Fanuc KAREL source: kb00086.KL

-- PROVISIONAL review KL for V770-1; original PC SHA256 901841f6cbabf7c2d2944ea3b2c585691836dcc631c9c3183b48748d21902244
-- Incomplete behavior may be omitted. Consult companion uncertainty JSON. Do not deploy.
PROGRAM KB00086
%NOLOCKGROUP
BEGIN
  -- UNRESOLVED_PC offsets 5-12; opcodes 9D,23
  -- UNRESOLVED_PC offsets 17-24; opcodes 9D,23
  -- UNRESOLVED_PC offsets 29-36; opcodes 9D,23
  -- UNRESOLVED_PC offsets 41-48; opcodes 9D,23
  -- UNRESOLVED_PC offsets 53-60; opcodes 9D,23
  -- UNRESOLVED_PC offsets 65-72; opcodes 9D,23
  -- UNRESOLVED_PC offsets 77-117; opcodes 27,22,22,22,22,22,22,31
  -- UNRESOLVED_PC offsets 122-126; opcodes 7F
END KB00086
